// TIA Portal V17 export
// export: Created 2025-03-07T09:23:49.8339125Z, ExportSetting WithDefaults, DisplayName Totally Integrated Automation Portal, DisplayVersion V17 Update 8, DisplayName TIA Portal Openness, DisplayVersion V17 Update 8, DisplayName TIA Portal Version Control Interface, DisplayVersion V17, DisplayName SINAMICS Startdrive Advanced, DisplayVersion V17 SP2, DisplayName SINAMICS Startdrive G110M, G120, G120C, G120D, G120P, G115D, DisplayVersion V17 SP2, DisplayName SINAMICS Startdrive G130, G150, S120, S150, SINAMICS MV, S210, DisplayVersion V17 SP2, DisplayName STEP 7 Professional, DisplayVersion V17 Update 8, DisplayName SINUMERIK ONE STEP 7 Toolbox, DisplayVersion V17 Update 12, DisplayName SINUMERIK 840D sl STEP 7 Toolbox, DisplayVersion V17 Update 12, DisplayName STEP 7 Safety, DisplayVersion V17 Update 6, DisplayName WinCC Advanced, DisplayVersion V17 Update 8
FUNCTION "FC7342_POWDER_TO_MACHINE_INTERLOCK" : Void   // FC7342, LAD
{ S7_Optimized_Access := 'TRUE' }
VERSION : 0.1
// stored: AutoNumber false, IsIECCheckEnabled false, SetENOAutomatically false, UDAEnableTagReadback false
BEGIN

REGION Network 1: LIFE BIT
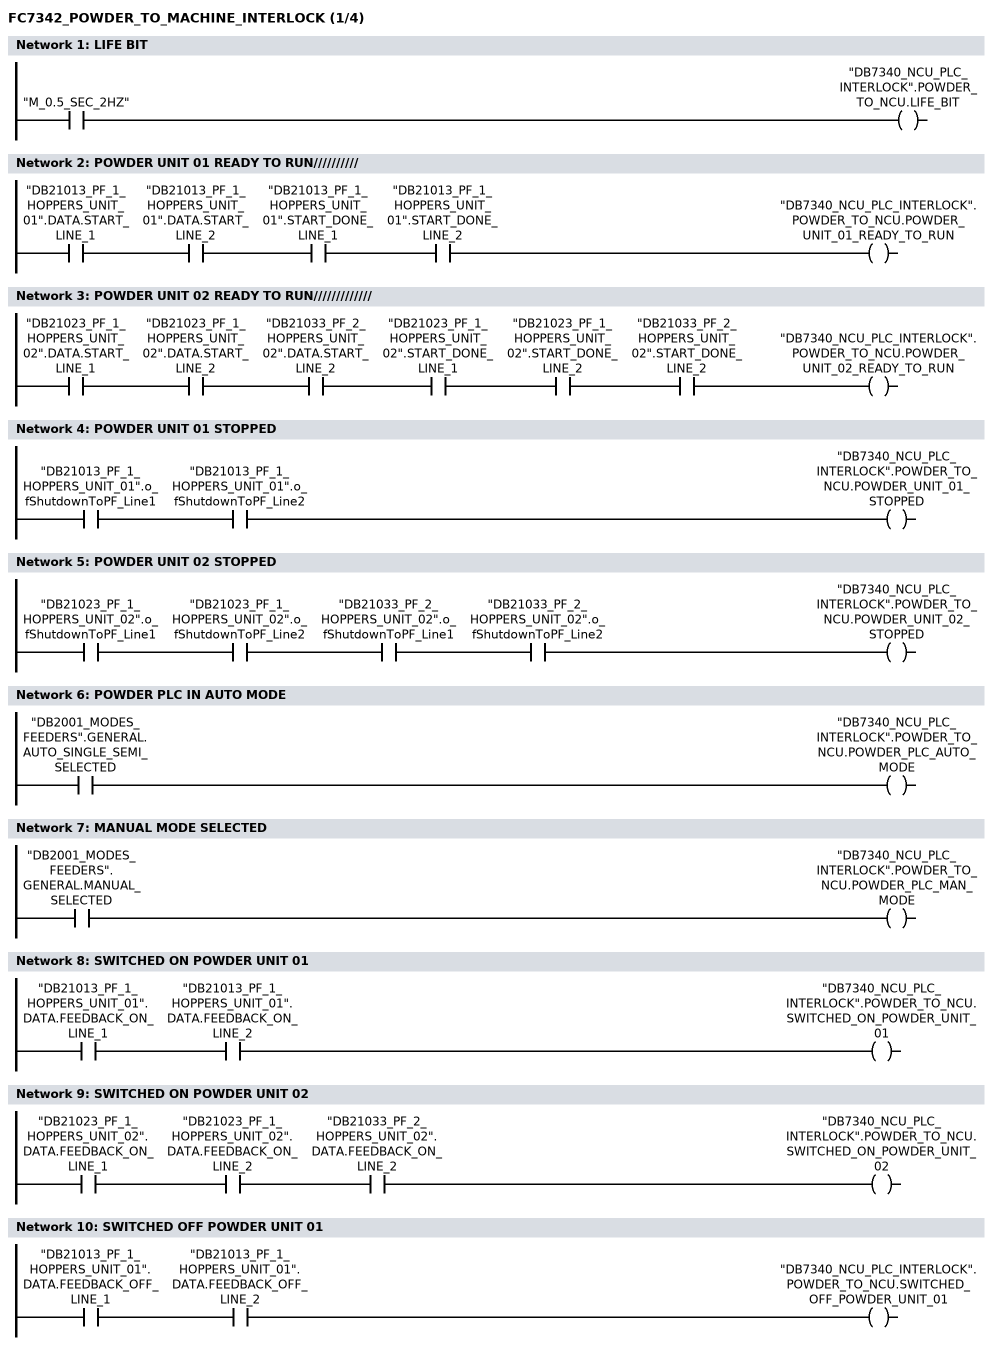
   RUNG wire#powerrail
      Contact( "M_0.5_SEC_2HZ" )
      Coil( "DB7340_NCU_PLC_INTERLOCK".POWDER_TO_NCU.LIFE_BIT )
   END_RUNG
   // the same network as SCL:
   "DB7340_NCU_PLC_INTERLOCK".POWDER_TO_NCU.LIFE_BIT := "M_0.5_SEC_2HZ";
END_REGION

REGION Network 2: POWDER UNIT 01 READY TO RUN//////////
   RUNG wire#powerrail
      Contact( "DB21013_PF_1_HOPPERS_UNIT_01".DATA.START_LINE_1 )
      Contact( "DB21013_PF_1_HOPPERS_UNIT_01".DATA.START_LINE_2 )
      Contact( "DB21013_PF_1_HOPPERS_UNIT_01".START_DONE_LINE_1 )
      Contact( "DB21013_PF_1_HOPPERS_UNIT_01".START_DONE_LINE_2 )
      Coil( "DB7340_NCU_PLC_INTERLOCK".POWDER_TO_NCU.POWDER_UNIT_01_READY_TO_RUN )
   END_RUNG
   // the same network as SCL:
   "DB7340_NCU_PLC_INTERLOCK".POWDER_TO_NCU.POWDER_UNIT_01_READY_TO_RUN := "DB21013_PF_1_HOPPERS_UNIT_01".DATA.START_LINE_1 AND "DB21013_PF_1_HOPPERS_UNIT_01".DATA.START_LINE_2 AND "DB21013_PF_1_HOPPERS_UNIT_01".START_DONE_LINE_1 AND "DB21013_PF_1_HOPPERS_UNIT_01".START_DONE_LINE_2;
END_REGION

REGION Network 3: POWDER UNIT 02 READY TO RUN/////////////
   RUNG wire#powerrail
      Contact( "DB21023_PF_1_HOPPERS_UNIT_02".DATA.START_LINE_1 )
      Contact( "DB21023_PF_1_HOPPERS_UNIT_02".DATA.START_LINE_2 )
      Contact( "DB21033_PF_2_HOPPERS_UNIT_02".DATA.START_LINE_2 )
      Contact( "DB21023_PF_1_HOPPERS_UNIT_02".START_DONE_LINE_1 )
      Contact( "DB21023_PF_1_HOPPERS_UNIT_02".START_DONE_LINE_2 )
      Contact( "DB21033_PF_2_HOPPERS_UNIT_02".START_DONE_LINE_2 )
      Coil( "DB7340_NCU_PLC_INTERLOCK".POWDER_TO_NCU.POWDER_UNIT_02_READY_TO_RUN )
   END_RUNG
   // the same network as SCL:
   "DB7340_NCU_PLC_INTERLOCK".POWDER_TO_NCU.POWDER_UNIT_02_READY_TO_RUN := "DB21023_PF_1_HOPPERS_UNIT_02".DATA.START_LINE_1 AND "DB21023_PF_1_HOPPERS_UNIT_02".DATA.START_LINE_2 AND "DB21033_PF_2_HOPPERS_UNIT_02".DATA.START_LINE_2 AND "DB21023_PF_1_HOPPERS_UNIT_02".START_DONE_LINE_1 AND "DB21023_PF_1_HOPPERS_UNIT_02".START_DONE_LINE_2 AND "DB21033_PF_2_HOPPERS_UNIT_02".START_DONE_LINE_2;
END_REGION

REGION Network 4: POWDER UNIT 01 STOPPED
   RUNG wire#powerrail
      Contact( "DB21013_PF_1_HOPPERS_UNIT_01".o_fShutdownToPF_Line1 )
      Contact( "DB21013_PF_1_HOPPERS_UNIT_01".o_fShutdownToPF_Line2 )
      Coil( "DB7340_NCU_PLC_INTERLOCK".POWDER_TO_NCU.POWDER_UNIT_01_STOPPED )
   END_RUNG
   // the same network as SCL:
   "DB7340_NCU_PLC_INTERLOCK".POWDER_TO_NCU.POWDER_UNIT_01_STOPPED := "DB21013_PF_1_HOPPERS_UNIT_01".o_fShutdownToPF_Line1 AND "DB21013_PF_1_HOPPERS_UNIT_01".o_fShutdownToPF_Line2;
END_REGION

REGION Network 5: POWDER UNIT 02 STOPPED
   RUNG wire#powerrail
      Contact( "DB21023_PF_1_HOPPERS_UNIT_02".o_fShutdownToPF_Line1 )
      Contact( "DB21023_PF_1_HOPPERS_UNIT_02".o_fShutdownToPF_Line2 )
      Contact( "DB21033_PF_2_HOPPERS_UNIT_02".o_fShutdownToPF_Line1 )
      Contact( "DB21033_PF_2_HOPPERS_UNIT_02".o_fShutdownToPF_Line2 )
      Coil( "DB7340_NCU_PLC_INTERLOCK".POWDER_TO_NCU.POWDER_UNIT_02_STOPPED )
   END_RUNG
   // the same network as SCL:
   "DB7340_NCU_PLC_INTERLOCK".POWDER_TO_NCU.POWDER_UNIT_02_STOPPED := "DB21023_PF_1_HOPPERS_UNIT_02".o_fShutdownToPF_Line1 AND "DB21023_PF_1_HOPPERS_UNIT_02".o_fShutdownToPF_Line2 AND "DB21033_PF_2_HOPPERS_UNIT_02".o_fShutdownToPF_Line1 AND "DB21033_PF_2_HOPPERS_UNIT_02".o_fShutdownToPF_Line2;
END_REGION

REGION Network 6: POWDER PLC IN AUTO MODE
   RUNG wire#powerrail
      Contact( "DB2001_MODES_FEEDERS".GENERAL.AUTO_SINGLE_SEMI_SELECTED )
      Coil( "DB7340_NCU_PLC_INTERLOCK".POWDER_TO_NCU.POWDER_PLC_AUTO_MODE )
   END_RUNG
   // the same network as SCL:
   "DB7340_NCU_PLC_INTERLOCK".POWDER_TO_NCU.POWDER_PLC_AUTO_MODE := "DB2001_MODES_FEEDERS".GENERAL.AUTO_SINGLE_SEMI_SELECTED;
END_REGION

REGION Network 7: MANUAL MODE SELECTED
   RUNG wire#powerrail
      Contact( "DB2001_MODES_FEEDERS".GENERAL.MANUAL_SELECTED )
      Coil( "DB7340_NCU_PLC_INTERLOCK".POWDER_TO_NCU.POWDER_PLC_MAN_MODE )
   END_RUNG
   // the same network as SCL:
   "DB7340_NCU_PLC_INTERLOCK".POWDER_TO_NCU.POWDER_PLC_MAN_MODE := "DB2001_MODES_FEEDERS".GENERAL.MANUAL_SELECTED;
END_REGION

REGION Network 8: SWITCHED ON POWDER UNIT 01
   RUNG wire#powerrail
      Contact( "DB21013_PF_1_HOPPERS_UNIT_01".DATA.FEEDBACK_ON_LINE_1 )
      Contact( "DB21013_PF_1_HOPPERS_UNIT_01".DATA.FEEDBACK_ON_LINE_2 )
      Coil( "DB7340_NCU_PLC_INTERLOCK".POWDER_TO_NCU.SWITCHED_ON_POWDER_UNIT_01 )
   END_RUNG
   // the same network as SCL:
   "DB7340_NCU_PLC_INTERLOCK".POWDER_TO_NCU.SWITCHED_ON_POWDER_UNIT_01 := "DB21013_PF_1_HOPPERS_UNIT_01".DATA.FEEDBACK_ON_LINE_1 AND "DB21013_PF_1_HOPPERS_UNIT_01".DATA.FEEDBACK_ON_LINE_2;
END_REGION

REGION Network 9: SWITCHED ON POWDER UNIT 02
   RUNG wire#powerrail
      Contact( "DB21023_PF_1_HOPPERS_UNIT_02".DATA.FEEDBACK_ON_LINE_1 )
      Contact( "DB21023_PF_1_HOPPERS_UNIT_02".DATA.FEEDBACK_ON_LINE_2 )
      Contact( "DB21033_PF_2_HOPPERS_UNIT_02".DATA.FEEDBACK_ON_LINE_2 )
      Coil( "DB7340_NCU_PLC_INTERLOCK".POWDER_TO_NCU.SWITCHED_ON_POWDER_UNIT_02 )
   END_RUNG
   // the same network as SCL:
   "DB7340_NCU_PLC_INTERLOCK".POWDER_TO_NCU.SWITCHED_ON_POWDER_UNIT_02 := "DB21023_PF_1_HOPPERS_UNIT_02".DATA.FEEDBACK_ON_LINE_1 AND "DB21023_PF_1_HOPPERS_UNIT_02".DATA.FEEDBACK_ON_LINE_2 AND "DB21033_PF_2_HOPPERS_UNIT_02".DATA.FEEDBACK_ON_LINE_2;
END_REGION

REGION Network 10: SWITCHED OFF POWDER UNIT 01
   RUNG wire#powerrail
      Contact( "DB21013_PF_1_HOPPERS_UNIT_01".DATA.FEEDBACK_OFF_LINE_1 )
      Contact( "DB21013_PF_1_HOPPERS_UNIT_01".DATA.FEEDBACK_OFF_LINE_2 )
      Coil( "DB7340_NCU_PLC_INTERLOCK".POWDER_TO_NCU.SWITCHED_OFF_POWDER_UNIT_01 )
   END_RUNG
   // the same network as SCL:
   "DB7340_NCU_PLC_INTERLOCK".POWDER_TO_NCU.SWITCHED_OFF_POWDER_UNIT_01 := "DB21013_PF_1_HOPPERS_UNIT_01".DATA.FEEDBACK_OFF_LINE_1 AND "DB21013_PF_1_HOPPERS_UNIT_01".DATA.FEEDBACK_OFF_LINE_2;
END_REGION

REGION Network 11: SWITCHED OFF POWDER UNIT 02
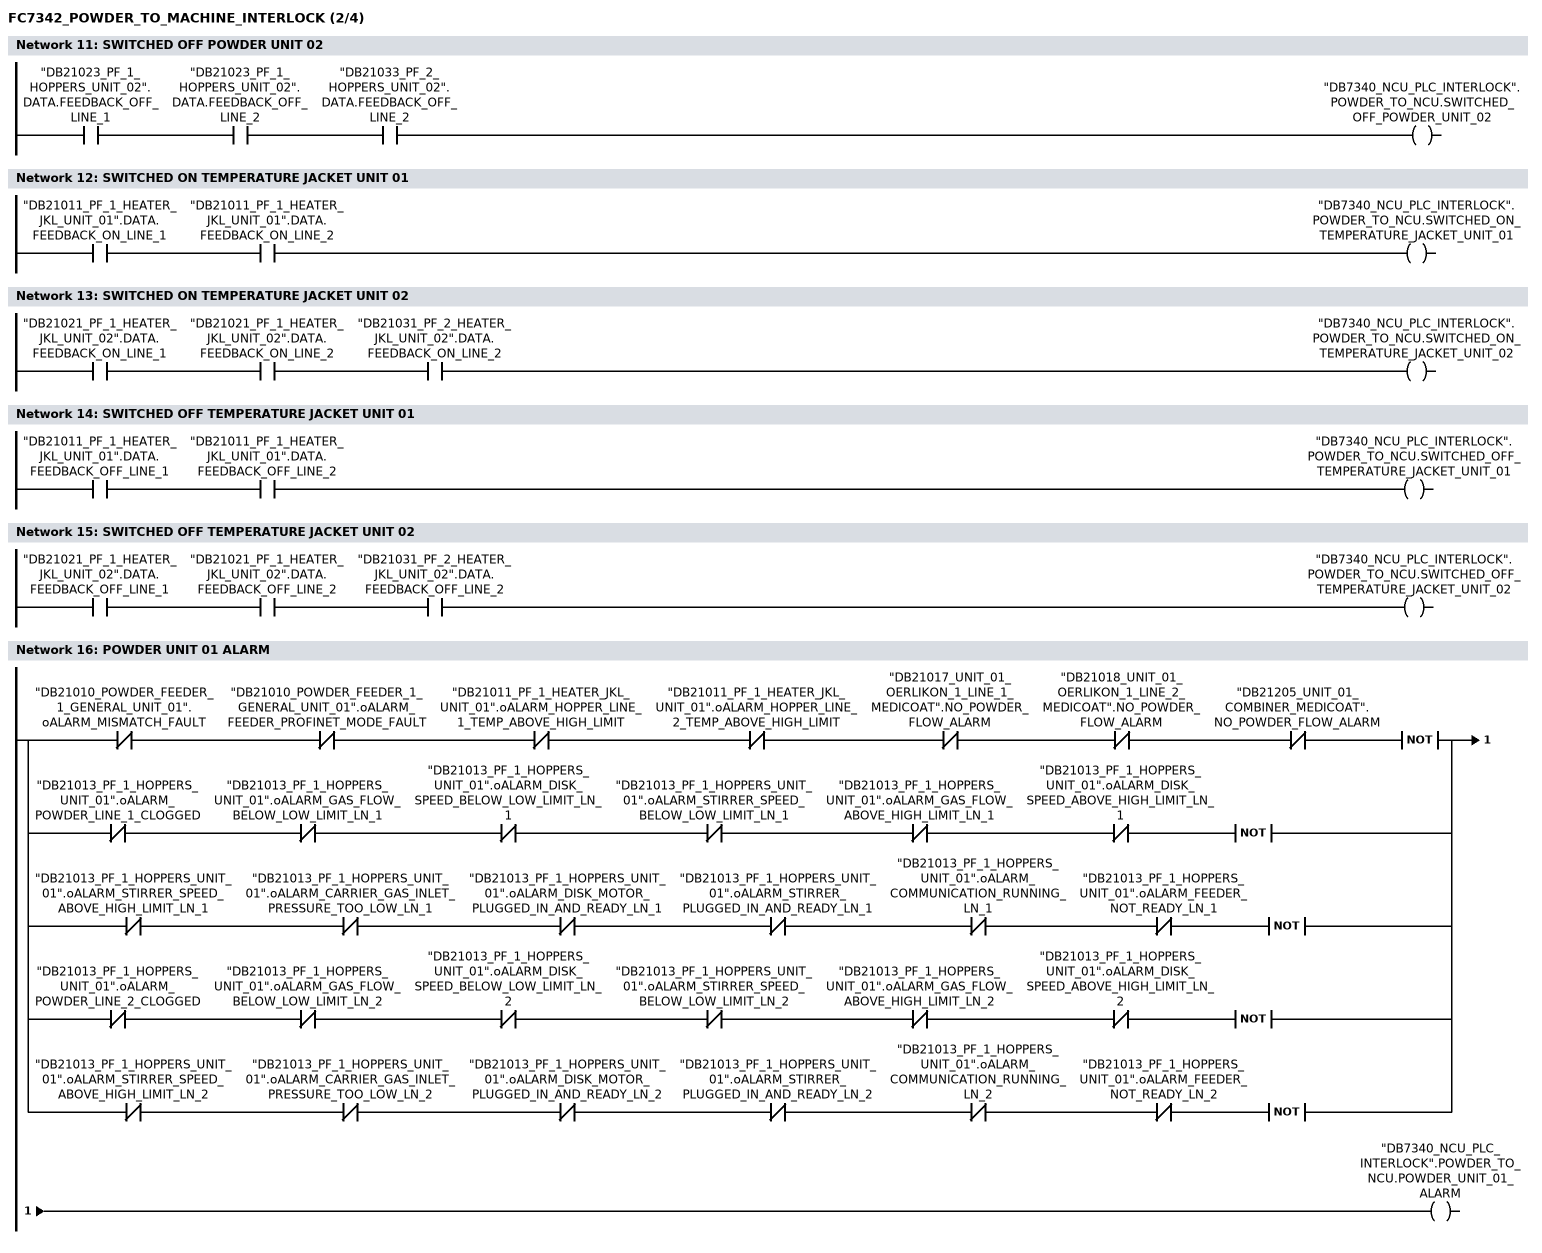
   RUNG wire#powerrail
      Contact( "DB21023_PF_1_HOPPERS_UNIT_02".DATA.FEEDBACK_OFF_LINE_1 )
      Contact( "DB21023_PF_1_HOPPERS_UNIT_02".DATA.FEEDBACK_OFF_LINE_2 )
      Contact( "DB21033_PF_2_HOPPERS_UNIT_02".DATA.FEEDBACK_OFF_LINE_2 )
      Coil( "DB7340_NCU_PLC_INTERLOCK".POWDER_TO_NCU.SWITCHED_OFF_POWDER_UNIT_02 )
   END_RUNG
   // the same network as SCL:
   "DB7340_NCU_PLC_INTERLOCK".POWDER_TO_NCU.SWITCHED_OFF_POWDER_UNIT_02 := "DB21023_PF_1_HOPPERS_UNIT_02".DATA.FEEDBACK_OFF_LINE_1 AND "DB21023_PF_1_HOPPERS_UNIT_02".DATA.FEEDBACK_OFF_LINE_2 AND "DB21033_PF_2_HOPPERS_UNIT_02".DATA.FEEDBACK_OFF_LINE_2;
END_REGION

REGION Network 12: SWITCHED ON TEMPERATURE JACKET UNIT 01
   RUNG wire#powerrail
      Contact( "DB21011_PF_1_HEATER_JKL_UNIT_01".DATA.FEEDBACK_ON_LINE_1 )
      Contact( "DB21011_PF_1_HEATER_JKL_UNIT_01".DATA.FEEDBACK_ON_LINE_2 )
      Coil( "DB7340_NCU_PLC_INTERLOCK".POWDER_TO_NCU.SWITCHED_ON_TEMPERATURE_JACKET_UNIT_01 )
   END_RUNG
   // the same network as SCL:
   "DB7340_NCU_PLC_INTERLOCK".POWDER_TO_NCU.SWITCHED_ON_TEMPERATURE_JACKET_UNIT_01 := "DB21011_PF_1_HEATER_JKL_UNIT_01".DATA.FEEDBACK_ON_LINE_1 AND "DB21011_PF_1_HEATER_JKL_UNIT_01".DATA.FEEDBACK_ON_LINE_2;
END_REGION

REGION Network 13: SWITCHED ON TEMPERATURE JACKET UNIT 02
   RUNG wire#powerrail
      Contact( "DB21021_PF_1_HEATER_JKL_UNIT_02".DATA.FEEDBACK_ON_LINE_1 )
      Contact( "DB21021_PF_1_HEATER_JKL_UNIT_02".DATA.FEEDBACK_ON_LINE_2 )
      Contact( "DB21031_PF_2_HEATER_JKL_UNIT_02".DATA.FEEDBACK_ON_LINE_2 )
      Coil( "DB7340_NCU_PLC_INTERLOCK".POWDER_TO_NCU.SWITCHED_ON_TEMPERATURE_JACKET_UNIT_02 )
   END_RUNG
   // the same network as SCL:
   "DB7340_NCU_PLC_INTERLOCK".POWDER_TO_NCU.SWITCHED_ON_TEMPERATURE_JACKET_UNIT_02 := "DB21021_PF_1_HEATER_JKL_UNIT_02".DATA.FEEDBACK_ON_LINE_1 AND "DB21021_PF_1_HEATER_JKL_UNIT_02".DATA.FEEDBACK_ON_LINE_2 AND "DB21031_PF_2_HEATER_JKL_UNIT_02".DATA.FEEDBACK_ON_LINE_2;
END_REGION

REGION Network 14: SWITCHED OFF TEMPERATURE JACKET UNIT 01
   RUNG wire#powerrail
      Contact( "DB21011_PF_1_HEATER_JKL_UNIT_01".DATA.FEEDBACK_OFF_LINE_1 )
      Contact( "DB21011_PF_1_HEATER_JKL_UNIT_01".DATA.FEEDBACK_OFF_LINE_2 )
      Coil( "DB7340_NCU_PLC_INTERLOCK".POWDER_TO_NCU.SWITCHED_OFF_TEMPERATURE_JACKET_UNIT_01 )
   END_RUNG
   // the same network as SCL:
   "DB7340_NCU_PLC_INTERLOCK".POWDER_TO_NCU.SWITCHED_OFF_TEMPERATURE_JACKET_UNIT_01 := "DB21011_PF_1_HEATER_JKL_UNIT_01".DATA.FEEDBACK_OFF_LINE_1 AND "DB21011_PF_1_HEATER_JKL_UNIT_01".DATA.FEEDBACK_OFF_LINE_2;
END_REGION

REGION Network 15: SWITCHED OFF TEMPERATURE JACKET UNIT 02
   RUNG wire#powerrail
      Contact( "DB21021_PF_1_HEATER_JKL_UNIT_02".DATA.FEEDBACK_OFF_LINE_1 )
      Contact( "DB21021_PF_1_HEATER_JKL_UNIT_02".DATA.FEEDBACK_OFF_LINE_2 )
      Contact( "DB21031_PF_2_HEATER_JKL_UNIT_02".DATA.FEEDBACK_OFF_LINE_2 )
      Coil( "DB7340_NCU_PLC_INTERLOCK".POWDER_TO_NCU.SWITCHED_OFF_TEMPERATURE_JACKET_UNIT_02 )
   END_RUNG
   // the same network as SCL:
   "DB7340_NCU_PLC_INTERLOCK".POWDER_TO_NCU.SWITCHED_OFF_TEMPERATURE_JACKET_UNIT_02 := "DB21021_PF_1_HEATER_JKL_UNIT_02".DATA.FEEDBACK_OFF_LINE_1 AND "DB21021_PF_1_HEATER_JKL_UNIT_02".DATA.FEEDBACK_OFF_LINE_2 AND "DB21031_PF_2_HEATER_JKL_UNIT_02".DATA.FEEDBACK_OFF_LINE_2;
END_REGION

REGION Network 16: POWDER UNIT 01 ALARM
   RUNG wire#powerrail
      I_Contact( "DB21010_POWDER_FEEDER_1_GENERAL_UNIT_01".oALARM_MISMATCH_FAULT )
      I_Contact( "DB21010_POWDER_FEEDER_1_GENERAL_UNIT_01".oALARM_FEEDER_PROFINET_MODE_FAULT )
      I_Contact( "DB21011_PF_1_HEATER_JKL_UNIT_01".oALARM_HOPPER_LINE_1_TEMP_ABOVE_HIGH_LIMIT )
      I_Contact( "DB21011_PF_1_HEATER_JKL_UNIT_01".oALARM_HOPPER_LINE_2_TEMP_ABOVE_HIGH_LIMIT )
      I_Contact( "DB21017_UNIT_01_OERLIKON_1_LINE_1_MEDICOAT".NO_POWDER_FLOW_ALARM )
      I_Contact( "DB21018_UNIT_01_OERLIKON_1_LINE_2_MEDICOAT".NO_POWDER_FLOW_ALARM )
      I_Contact( "DB21205_UNIT_01_COMBINER_MEDICOAT".NO_POWDER_FLOW_ALARM )
      Not()
      wire#w1
      Coil( "DB7340_NCU_PLC_INTERLOCK".POWDER_TO_NCU.POWDER_UNIT_01_ALARM )
   END_RUNG
   RUNG wire#powerrail
      I_Contact( "DB21013_PF_1_HOPPERS_UNIT_01".oALARM_POWDER_LINE_1_CLOGGED )
      I_Contact( "DB21013_PF_1_HOPPERS_UNIT_01".oALARM_GAS_FLOW_BELOW_LOW_LIMIT_LN_1 )
      I_Contact( "DB21013_PF_1_HOPPERS_UNIT_01".oALARM_DISK_SPEED_BELOW_LOW_LIMIT_LN_1 )
      I_Contact( "DB21013_PF_1_HOPPERS_UNIT_01".oALARM_STIRRER_SPEED_BELOW_LOW_LIMIT_LN_1 )
      I_Contact( "DB21013_PF_1_HOPPERS_UNIT_01".oALARM_GAS_FLOW_ABOVE_HIGH_LIMIT_LN_1 )
      I_Contact( "DB21013_PF_1_HOPPERS_UNIT_01".oALARM_DISK_SPEED_ABOVE_HIGH_LIMIT_LN_1 )
      Not()
   END_RUNG wire#w1
   RUNG wire#powerrail
      I_Contact( "DB21013_PF_1_HOPPERS_UNIT_01".oALARM_STIRRER_SPEED_ABOVE_HIGH_LIMIT_LN_1 )
      I_Contact( "DB21013_PF_1_HOPPERS_UNIT_01".oALARM_CARRIER_GAS_INLET_PRESSURE_TOO_LOW_LN_1 )
      I_Contact( "DB21013_PF_1_HOPPERS_UNIT_01".oALARM_DISK_MOTOR_PLUGGED_IN_AND_READY_LN_1 )
      I_Contact( "DB21013_PF_1_HOPPERS_UNIT_01".oALARM_STIRRER_PLUGGED_IN_AND_READY_LN_1 )
      I_Contact( "DB21013_PF_1_HOPPERS_UNIT_01".oALARM_COMMUNICATION_RUNNING_LN_1 )
      I_Contact( "DB21013_PF_1_HOPPERS_UNIT_01".oALARM_FEEDER_NOT_READY_LN_1 )
      Not()
   END_RUNG wire#w1
   RUNG wire#powerrail
      I_Contact( "DB21013_PF_1_HOPPERS_UNIT_01".oALARM_POWDER_LINE_2_CLOGGED )
      I_Contact( "DB21013_PF_1_HOPPERS_UNIT_01".oALARM_GAS_FLOW_BELOW_LOW_LIMIT_LN_2 )
      I_Contact( "DB21013_PF_1_HOPPERS_UNIT_01".oALARM_DISK_SPEED_BELOW_LOW_LIMIT_LN_2 )
      I_Contact( "DB21013_PF_1_HOPPERS_UNIT_01".oALARM_STIRRER_SPEED_BELOW_LOW_LIMIT_LN_2 )
      I_Contact( "DB21013_PF_1_HOPPERS_UNIT_01".oALARM_GAS_FLOW_ABOVE_HIGH_LIMIT_LN_2 )
      I_Contact( "DB21013_PF_1_HOPPERS_UNIT_01".oALARM_DISK_SPEED_ABOVE_HIGH_LIMIT_LN_2 )
      Not()
   END_RUNG wire#w1
   RUNG wire#powerrail
      I_Contact( "DB21013_PF_1_HOPPERS_UNIT_01".oALARM_STIRRER_SPEED_ABOVE_HIGH_LIMIT_LN_2 )
      I_Contact( "DB21013_PF_1_HOPPERS_UNIT_01".oALARM_CARRIER_GAS_INLET_PRESSURE_TOO_LOW_LN_2 )
      I_Contact( "DB21013_PF_1_HOPPERS_UNIT_01".oALARM_DISK_MOTOR_PLUGGED_IN_AND_READY_LN_2 )
      I_Contact( "DB21013_PF_1_HOPPERS_UNIT_01".oALARM_STIRRER_PLUGGED_IN_AND_READY_LN_2 )
      I_Contact( "DB21013_PF_1_HOPPERS_UNIT_01".oALARM_COMMUNICATION_RUNNING_LN_2 )
      I_Contact( "DB21013_PF_1_HOPPERS_UNIT_01".oALARM_FEEDER_NOT_READY_LN_2 )
      Not()
   END_RUNG wire#w1
   // the same network as SCL:
   "DB7340_NCU_PLC_INTERLOCK".POWDER_TO_NCU.POWDER_UNIT_01_ALARM := NOT (NOT "DB21010_POWDER_FEEDER_1_GENERAL_UNIT_01".oALARM_MISMATCH_FAULT AND NOT "DB21010_POWDER_FEEDER_1_GENERAL_UNIT_01".oALARM_FEEDER_PROFINET_MODE_FAULT AND NOT "DB21011_PF_1_HEATER_JKL_UNIT_01".oALARM_HOPPER_LINE_1_TEMP_ABOVE_HIGH_LIMIT AND NOT "DB21011_PF_1_HEATER_JKL_UNIT_01".oALARM_HOPPER_LINE_2_TEMP_ABOVE_HIGH_LIMIT AND NOT "DB21017_UNIT_01_OERLIKON_1_LINE_1_MEDICOAT".NO_POWDER_FLOW_ALARM AND NOT "DB21018_UNIT_01_OERLIKON_1_LINE_2_MEDICOAT".NO_POWDER_FLOW_ALARM AND NOT "DB21205_UNIT_01_COMBINER_MEDICOAT".NO_POWDER_FLOW_ALARM) OR NOT (NOT "DB21013_PF_1_HOPPERS_UNIT_01".oALARM_POWDER_LINE_1_CLOGGED AND NOT "DB21013_PF_1_HOPPERS_UNIT_01".oALARM_GAS_FLOW_BELOW_LOW_LIMIT_LN_1 AND NOT "DB21013_PF_1_HOPPERS_UNIT_01".oALARM_DISK_SPEED_BELOW_LOW_LIMIT_LN_1 AND NOT "DB21013_PF_1_HOPPERS_UNIT_01".oALARM_STIRRER_SPEED_BELOW_LOW_LIMIT_LN_1 AND NOT "DB21013_PF_1_HOPPERS_UNIT_01".oALARM_GAS_FLOW_ABOVE_HIGH_LIMIT_LN_1 AND NOT "DB21013_PF_1_HOPPERS_UNIT_01".oALARM_DISK_SPEED_ABOVE_HIGH_LIMIT_LN_1) OR NOT (NOT "DB21013_PF_1_HOPPERS_UNIT_01".oALARM_STIRRER_SPEED_ABOVE_HIGH_LIMIT_LN_1 AND NOT "DB21013_PF_1_HOPPERS_UNIT_01".oALARM_CARRIER_GAS_INLET_PRESSURE_TOO_LOW_LN_1 AND NOT "DB21013_PF_1_HOPPERS_UNIT_01".oALARM_DISK_MOTOR_PLUGGED_IN_AND_READY_LN_1 AND NOT "DB21013_PF_1_HOPPERS_UNIT_01".oALARM_STIRRER_PLUGGED_IN_AND_READY_LN_1 AND NOT "DB21013_PF_1_HOPPERS_UNIT_01".oALARM_COMMUNICATION_RUNNING_LN_1 AND NOT "DB21013_PF_1_HOPPERS_UNIT_01".oALARM_FEEDER_NOT_READY_LN_1) OR NOT (NOT "DB21013_PF_1_HOPPERS_UNIT_01".oALARM_POWDER_LINE_2_CLOGGED AND NOT "DB21013_PF_1_HOPPERS_UNIT_01".oALARM_GAS_FLOW_BELOW_LOW_LIMIT_LN_2 AND NOT "DB21013_PF_1_HOPPERS_UNIT_01".oALARM_DISK_SPEED_BELOW_LOW_LIMIT_LN_2 AND NOT "DB21013_PF_1_HOPPERS_UNIT_01".oALARM_STIRRER_SPEED_BELOW_LOW_LIMIT_LN_2 AND NOT "DB21013_PF_1_HOPPERS_UNIT_01".oALARM_GAS_FLOW_ABOVE_HIGH_LIMIT_LN_2 AND NOT "DB21013_PF_1_HOPPERS_UNIT_01".oALARM_DISK_SPEED_ABOVE_HIGH_LIMIT_LN_2) OR NOT (NOT "DB21013_PF_1_HOPPERS_UNIT_01".oALARM_STIRRER_SPEED_ABOVE_HIGH_LIMIT_LN_2 AND NOT "DB21013_PF_1_HOPPERS_UNIT_01".oALARM_CARRIER_GAS_INLET_PRESSURE_TOO_LOW_LN_2 AND NOT "DB21013_PF_1_HOPPERS_UNIT_01".oALARM_DISK_MOTOR_PLUGGED_IN_AND_READY_LN_2 AND NOT "DB21013_PF_1_HOPPERS_UNIT_01".oALARM_STIRRER_PLUGGED_IN_AND_READY_LN_2 AND NOT "DB21013_PF_1_HOPPERS_UNIT_01".oALARM_COMMUNICATION_RUNNING_LN_2 AND NOT "DB21013_PF_1_HOPPERS_UNIT_01".oALARM_FEEDER_NOT_READY_LN_2);
END_REGION

REGION Network 17: POWDER UNIT 02 ALARM
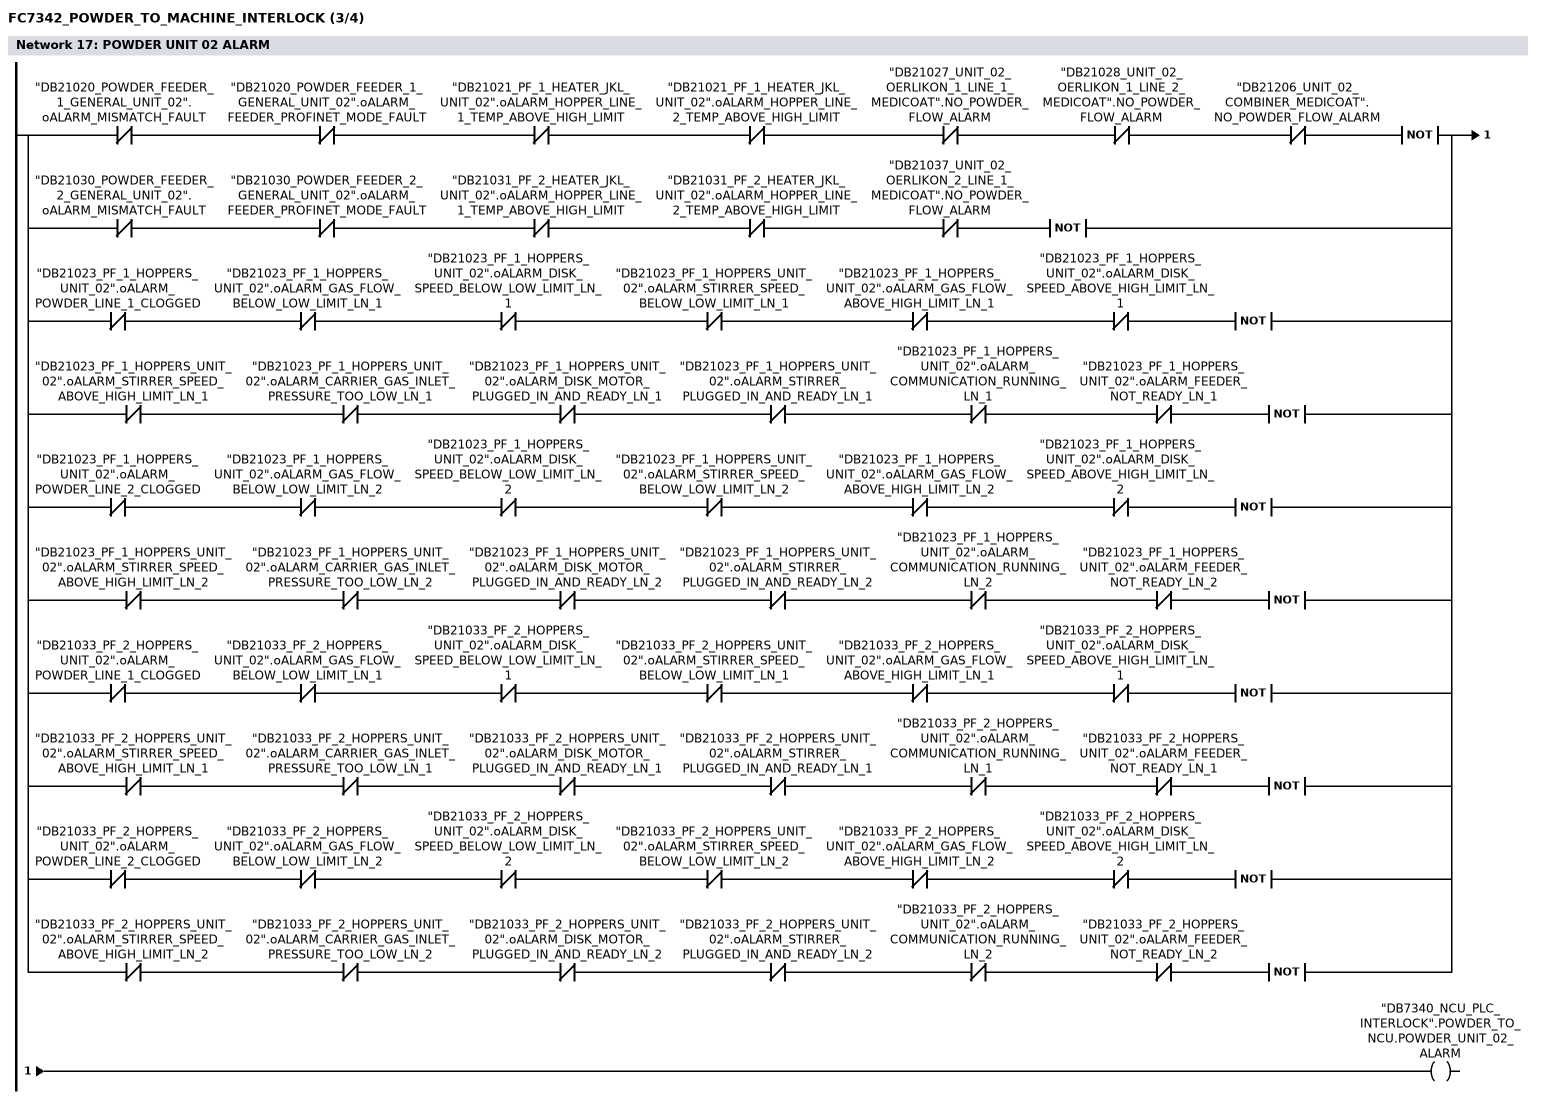
   RUNG wire#powerrail
      I_Contact( "DB21020_POWDER_FEEDER_1_GENERAL_UNIT_02".oALARM_MISMATCH_FAULT )
      I_Contact( "DB21020_POWDER_FEEDER_1_GENERAL_UNIT_02".oALARM_FEEDER_PROFINET_MODE_FAULT )
      I_Contact( "DB21021_PF_1_HEATER_JKL_UNIT_02".oALARM_HOPPER_LINE_1_TEMP_ABOVE_HIGH_LIMIT )
      I_Contact( "DB21021_PF_1_HEATER_JKL_UNIT_02".oALARM_HOPPER_LINE_2_TEMP_ABOVE_HIGH_LIMIT )
      I_Contact( "DB21027_UNIT_02_OERLIKON_1_LINE_1_MEDICOAT".NO_POWDER_FLOW_ALARM )
      I_Contact( "DB21028_UNIT_02_OERLIKON_1_LINE_2_MEDICOAT".NO_POWDER_FLOW_ALARM )
      I_Contact( "DB21206_UNIT_02_COMBINER_MEDICOAT".NO_POWDER_FLOW_ALARM )
      Not()
      wire#w1
      Coil( "DB7340_NCU_PLC_INTERLOCK".POWDER_TO_NCU.POWDER_UNIT_02_ALARM )
   END_RUNG
   RUNG wire#powerrail
      I_Contact( "DB21030_POWDER_FEEDER_2_GENERAL_UNIT_02".oALARM_MISMATCH_FAULT )
      I_Contact( "DB21030_POWDER_FEEDER_2_GENERAL_UNIT_02".oALARM_FEEDER_PROFINET_MODE_FAULT )
      I_Contact( "DB21031_PF_2_HEATER_JKL_UNIT_02".oALARM_HOPPER_LINE_1_TEMP_ABOVE_HIGH_LIMIT )
      I_Contact( "DB21031_PF_2_HEATER_JKL_UNIT_02".oALARM_HOPPER_LINE_2_TEMP_ABOVE_HIGH_LIMIT )
      I_Contact( "DB21037_UNIT_02_OERLIKON_2_LINE_1_MEDICOAT".NO_POWDER_FLOW_ALARM )
      Not()
   END_RUNG wire#w1
   RUNG wire#powerrail
      I_Contact( "DB21023_PF_1_HOPPERS_UNIT_02".oALARM_POWDER_LINE_1_CLOGGED )
      I_Contact( "DB21023_PF_1_HOPPERS_UNIT_02".oALARM_GAS_FLOW_BELOW_LOW_LIMIT_LN_1 )
      I_Contact( "DB21023_PF_1_HOPPERS_UNIT_02".oALARM_DISK_SPEED_BELOW_LOW_LIMIT_LN_1 )
      I_Contact( "DB21023_PF_1_HOPPERS_UNIT_02".oALARM_STIRRER_SPEED_BELOW_LOW_LIMIT_LN_1 )
      I_Contact( "DB21023_PF_1_HOPPERS_UNIT_02".oALARM_GAS_FLOW_ABOVE_HIGH_LIMIT_LN_1 )
      I_Contact( "DB21023_PF_1_HOPPERS_UNIT_02".oALARM_DISK_SPEED_ABOVE_HIGH_LIMIT_LN_1 )
      Not()
   END_RUNG wire#w1
   RUNG wire#powerrail
      I_Contact( "DB21023_PF_1_HOPPERS_UNIT_02".oALARM_STIRRER_SPEED_ABOVE_HIGH_LIMIT_LN_1 )
      I_Contact( "DB21023_PF_1_HOPPERS_UNIT_02".oALARM_CARRIER_GAS_INLET_PRESSURE_TOO_LOW_LN_1 )
      I_Contact( "DB21023_PF_1_HOPPERS_UNIT_02".oALARM_DISK_MOTOR_PLUGGED_IN_AND_READY_LN_1 )
      I_Contact( "DB21023_PF_1_HOPPERS_UNIT_02".oALARM_STIRRER_PLUGGED_IN_AND_READY_LN_1 )
      I_Contact( "DB21023_PF_1_HOPPERS_UNIT_02".oALARM_COMMUNICATION_RUNNING_LN_1 )
      I_Contact( "DB21023_PF_1_HOPPERS_UNIT_02".oALARM_FEEDER_NOT_READY_LN_1 )
      Not()
   END_RUNG wire#w1
   RUNG wire#powerrail
      I_Contact( "DB21023_PF_1_HOPPERS_UNIT_02".oALARM_POWDER_LINE_2_CLOGGED )
      I_Contact( "DB21023_PF_1_HOPPERS_UNIT_02".oALARM_GAS_FLOW_BELOW_LOW_LIMIT_LN_2 )
      I_Contact( "DB21023_PF_1_HOPPERS_UNIT_02".oALARM_DISK_SPEED_BELOW_LOW_LIMIT_LN_2 )
      I_Contact( "DB21023_PF_1_HOPPERS_UNIT_02".oALARM_STIRRER_SPEED_BELOW_LOW_LIMIT_LN_2 )
      I_Contact( "DB21023_PF_1_HOPPERS_UNIT_02".oALARM_GAS_FLOW_ABOVE_HIGH_LIMIT_LN_2 )
      I_Contact( "DB21023_PF_1_HOPPERS_UNIT_02".oALARM_DISK_SPEED_ABOVE_HIGH_LIMIT_LN_2 )
      Not()
   END_RUNG wire#w1
   RUNG wire#powerrail
      I_Contact( "DB21023_PF_1_HOPPERS_UNIT_02".oALARM_STIRRER_SPEED_ABOVE_HIGH_LIMIT_LN_2 )
      I_Contact( "DB21023_PF_1_HOPPERS_UNIT_02".oALARM_CARRIER_GAS_INLET_PRESSURE_TOO_LOW_LN_2 )
      I_Contact( "DB21023_PF_1_HOPPERS_UNIT_02".oALARM_DISK_MOTOR_PLUGGED_IN_AND_READY_LN_2 )
      I_Contact( "DB21023_PF_1_HOPPERS_UNIT_02".oALARM_STIRRER_PLUGGED_IN_AND_READY_LN_2 )
      I_Contact( "DB21023_PF_1_HOPPERS_UNIT_02".oALARM_COMMUNICATION_RUNNING_LN_2 )
      I_Contact( "DB21023_PF_1_HOPPERS_UNIT_02".oALARM_FEEDER_NOT_READY_LN_2 )
      Not()
   END_RUNG wire#w1
   RUNG wire#powerrail
      I_Contact( "DB21033_PF_2_HOPPERS_UNIT_02".oALARM_POWDER_LINE_1_CLOGGED )
      I_Contact( "DB21033_PF_2_HOPPERS_UNIT_02".oALARM_GAS_FLOW_BELOW_LOW_LIMIT_LN_1 )
      I_Contact( "DB21033_PF_2_HOPPERS_UNIT_02".oALARM_DISK_SPEED_BELOW_LOW_LIMIT_LN_1 )
      I_Contact( "DB21033_PF_2_HOPPERS_UNIT_02".oALARM_STIRRER_SPEED_BELOW_LOW_LIMIT_LN_1 )
      I_Contact( "DB21033_PF_2_HOPPERS_UNIT_02".oALARM_GAS_FLOW_ABOVE_HIGH_LIMIT_LN_1 )
      I_Contact( "DB21033_PF_2_HOPPERS_UNIT_02".oALARM_DISK_SPEED_ABOVE_HIGH_LIMIT_LN_1 )
      Not()
   END_RUNG wire#w1
   RUNG wire#powerrail
      I_Contact( "DB21033_PF_2_HOPPERS_UNIT_02".oALARM_STIRRER_SPEED_ABOVE_HIGH_LIMIT_LN_1 )
      I_Contact( "DB21033_PF_2_HOPPERS_UNIT_02".oALARM_CARRIER_GAS_INLET_PRESSURE_TOO_LOW_LN_1 )
      I_Contact( "DB21033_PF_2_HOPPERS_UNIT_02".oALARM_DISK_MOTOR_PLUGGED_IN_AND_READY_LN_1 )
      I_Contact( "DB21033_PF_2_HOPPERS_UNIT_02".oALARM_STIRRER_PLUGGED_IN_AND_READY_LN_1 )
      I_Contact( "DB21033_PF_2_HOPPERS_UNIT_02".oALARM_COMMUNICATION_RUNNING_LN_1 )
      I_Contact( "DB21033_PF_2_HOPPERS_UNIT_02".oALARM_FEEDER_NOT_READY_LN_1 )
      Not()
   END_RUNG wire#w1
   RUNG wire#powerrail
      I_Contact( "DB21033_PF_2_HOPPERS_UNIT_02".oALARM_POWDER_LINE_2_CLOGGED )
      I_Contact( "DB21033_PF_2_HOPPERS_UNIT_02".oALARM_GAS_FLOW_BELOW_LOW_LIMIT_LN_2 )
      I_Contact( "DB21033_PF_2_HOPPERS_UNIT_02".oALARM_DISK_SPEED_BELOW_LOW_LIMIT_LN_2 )
      I_Contact( "DB21033_PF_2_HOPPERS_UNIT_02".oALARM_STIRRER_SPEED_BELOW_LOW_LIMIT_LN_2 )
      I_Contact( "DB21033_PF_2_HOPPERS_UNIT_02".oALARM_GAS_FLOW_ABOVE_HIGH_LIMIT_LN_2 )
      I_Contact( "DB21033_PF_2_HOPPERS_UNIT_02".oALARM_DISK_SPEED_ABOVE_HIGH_LIMIT_LN_2 )
      Not()
   END_RUNG wire#w1
   RUNG wire#powerrail
      I_Contact( "DB21033_PF_2_HOPPERS_UNIT_02".oALARM_STIRRER_SPEED_ABOVE_HIGH_LIMIT_LN_2 )
      I_Contact( "DB21033_PF_2_HOPPERS_UNIT_02".oALARM_CARRIER_GAS_INLET_PRESSURE_TOO_LOW_LN_2 )
      I_Contact( "DB21033_PF_2_HOPPERS_UNIT_02".oALARM_DISK_MOTOR_PLUGGED_IN_AND_READY_LN_2 )
      I_Contact( "DB21033_PF_2_HOPPERS_UNIT_02".oALARM_STIRRER_PLUGGED_IN_AND_READY_LN_2 )
      I_Contact( "DB21033_PF_2_HOPPERS_UNIT_02".oALARM_COMMUNICATION_RUNNING_LN_2 )
      I_Contact( "DB21033_PF_2_HOPPERS_UNIT_02".oALARM_FEEDER_NOT_READY_LN_2 )
      Not()
   END_RUNG wire#w1
   // the same network as SCL:
   "DB7340_NCU_PLC_INTERLOCK".POWDER_TO_NCU.POWDER_UNIT_02_ALARM := NOT (NOT "DB21020_POWDER_FEEDER_1_GENERAL_UNIT_02".oALARM_MISMATCH_FAULT AND NOT "DB21020_POWDER_FEEDER_1_GENERAL_UNIT_02".oALARM_FEEDER_PROFINET_MODE_FAULT AND NOT "DB21021_PF_1_HEATER_JKL_UNIT_02".oALARM_HOPPER_LINE_1_TEMP_ABOVE_HIGH_LIMIT AND NOT "DB21021_PF_1_HEATER_JKL_UNIT_02".oALARM_HOPPER_LINE_2_TEMP_ABOVE_HIGH_LIMIT AND NOT "DB21027_UNIT_02_OERLIKON_1_LINE_1_MEDICOAT".NO_POWDER_FLOW_ALARM AND NOT "DB21028_UNIT_02_OERLIKON_1_LINE_2_MEDICOAT".NO_POWDER_FLOW_ALARM AND NOT "DB21206_UNIT_02_COMBINER_MEDICOAT".NO_POWDER_FLOW_ALARM) OR NOT (NOT "DB21030_POWDER_FEEDER_2_GENERAL_UNIT_02".oALARM_MISMATCH_FAULT AND NOT "DB21030_POWDER_FEEDER_2_GENERAL_UNIT_02".oALARM_FEEDER_PROFINET_MODE_FAULT AND NOT "DB21031_PF_2_HEATER_JKL_UNIT_02".oALARM_HOPPER_LINE_1_TEMP_ABOVE_HIGH_LIMIT AND NOT "DB21031_PF_2_HEATER_JKL_UNIT_02".oALARM_HOPPER_LINE_2_TEMP_ABOVE_HIGH_LIMIT AND NOT "DB21037_UNIT_02_OERLIKON_2_LINE_1_MEDICOAT".NO_POWDER_FLOW_ALARM) OR NOT (NOT "DB21023_PF_1_HOPPERS_UNIT_02".oALARM_POWDER_LINE_1_CLOGGED AND NOT "DB21023_PF_1_HOPPERS_UNIT_02".oALARM_GAS_FLOW_BELOW_LOW_LIMIT_LN_1 AND NOT "DB21023_PF_1_HOPPERS_UNIT_02".oALARM_DISK_SPEED_BELOW_LOW_LIMIT_LN_1 AND NOT "DB21023_PF_1_HOPPERS_UNIT_02".oALARM_STIRRER_SPEED_BELOW_LOW_LIMIT_LN_1 AND NOT "DB21023_PF_1_HOPPERS_UNIT_02".oALARM_GAS_FLOW_ABOVE_HIGH_LIMIT_LN_1 AND NOT "DB21023_PF_1_HOPPERS_UNIT_02".oALARM_DISK_SPEED_ABOVE_HIGH_LIMIT_LN_1) OR NOT (NOT "DB21023_PF_1_HOPPERS_UNIT_02".oALARM_STIRRER_SPEED_ABOVE_HIGH_LIMIT_LN_1 AND NOT "DB21023_PF_1_HOPPERS_UNIT_02".oALARM_CARRIER_GAS_INLET_PRESSURE_TOO_LOW_LN_1 AND NOT "DB21023_PF_1_HOPPERS_UNIT_02".oALARM_DISK_MOTOR_PLUGGED_IN_AND_READY_LN_1 AND NOT "DB21023_PF_1_HOPPERS_UNIT_02".oALARM_STIRRER_PLUGGED_IN_AND_READY_LN_1 AND NOT "DB21023_PF_1_HOPPERS_UNIT_02".oALARM_COMMUNICATION_RUNNING_LN_1 AND NOT "DB21023_PF_1_HOPPERS_UNIT_02".oALARM_FEEDER_NOT_READY_LN_1) OR NOT (NOT "DB21023_PF_1_HOPPERS_UNIT_02".oALARM_POWDER_LINE_2_CLOGGED AND NOT "DB21023_PF_1_HOPPERS_UNIT_02".oALARM_GAS_FLOW_BELOW_LOW_LIMIT_LN_2 AND NOT "DB21023_PF_1_HOPPERS_UNIT_02".oALARM_DISK_SPEED_BELOW_LOW_LIMIT_LN_2 AND NOT "DB21023_PF_1_HOPPERS_UNIT_02".oALARM_STIRRER_SPEED_BELOW_LOW_LIMIT_LN_2 AND NOT "DB21023_PF_1_HOPPERS_UNIT_02".oALARM_GAS_FLOW_ABOVE_HIGH_LIMIT_LN_2 AND NOT "DB21023_PF_1_HOPPERS_UNIT_02".oALARM_DISK_SPEED_ABOVE_HIGH_LIMIT_LN_2) OR NOT (NOT "DB21023_PF_1_HOPPERS_UNIT_02".oALARM_STIRRER_SPEED_ABOVE_HIGH_LIMIT_LN_2 AND NOT "DB21023_PF_1_HOPPERS_UNIT_02".oALARM_CARRIER_GAS_INLET_PRESSURE_TOO_LOW_LN_2 AND NOT "DB21023_PF_1_HOPPERS_UNIT_02".oALARM_DISK_MOTOR_PLUGGED_IN_AND_READY_LN_2 AND NOT "DB21023_PF_1_HOPPERS_UNIT_02".oALARM_STIRRER_PLUGGED_IN_AND_READY_LN_2 AND NOT "DB21023_PF_1_HOPPERS_UNIT_02".oALARM_COMMUNICATION_RUNNING_LN_2 AND NOT "DB21023_PF_1_HOPPERS_UNIT_02".oALARM_FEEDER_NOT_READY_LN_2) OR NOT (NOT "DB21033_PF_2_HOPPERS_UNIT_02".oALARM_POWDER_LINE_1_CLOGGED AND NOT "DB21033_PF_2_HOPPERS_UNIT_02".oALARM_GAS_FLOW_BELOW_LOW_LIMIT_LN_1 AND NOT "DB21033_PF_2_HOPPERS_UNIT_02".oALARM_DISK_SPEED_BELOW_LOW_LIMIT_LN_1 AND NOT "DB21033_PF_2_HOPPERS_UNIT_02".oALARM_STIRRER_SPEED_BELOW_LOW_LIMIT_LN_1 AND NOT "DB21033_PF_2_HOPPERS_UNIT_02".oALARM_GAS_FLOW_ABOVE_HIGH_LIMIT_LN_1 AND NOT "DB21033_PF_2_HOPPERS_UNIT_02".oALARM_DISK_SPEED_ABOVE_HIGH_LIMIT_LN_1) OR NOT (NOT "DB21033_PF_2_HOPPERS_UNIT_02".oALARM_STIRRER_SPEED_ABOVE_HIGH_LIMIT_LN_1 AND NOT "DB21033_PF_2_HOPPERS_UNIT_02".oALARM_CARRIER_GAS_INLET_PRESSURE_TOO_LOW_LN_1 AND NOT "DB21033_PF_2_HOPPERS_UNIT_02".oALARM_DISK_MOTOR_PLUGGED_IN_AND_READY_LN_1 AND NOT "DB21033_PF_2_HOPPERS_UNIT_02".oALARM_STIRRER_PLUGGED_IN_AND_READY_LN_1 AND NOT "DB21033_PF_2_HOPPERS_UNIT_02".oALARM_COMMUNICATION_RUNNING_LN_1 AND NOT "DB21033_PF_2_HOPPERS_UNIT_02".oALARM_FEEDER_NOT_READY_LN_1) OR NOT (NOT "DB21033_PF_2_HOPPERS_UNIT_02".oALARM_POWDER_LINE_2_CLOGGED AND NOT "DB21033_PF_2_HOPPERS_UNIT_02".oALARM_GAS_FLOW_BELOW_LOW_LIMIT_LN_2 AND NOT "DB21033_PF_2_HOPPERS_UNIT_02".oALARM_DISK_SPEED_BELOW_LOW_LIMIT_LN_2 AND NOT "DB21033_PF_2_HOPPERS_UNIT_02".oALARM_STIRRER_SPEED_BELOW_LOW_LIMIT_LN_2 AND NOT "DB21033_PF_2_HOPPERS_UNIT_02".oALARM_GAS_FLOW_ABOVE_HIGH_LIMIT_LN_2 AND NOT "DB21033_PF_2_HOPPERS_UNIT_02".oALARM_DISK_SPEED_ABOVE_HIGH_LIMIT_LN_2) OR NOT (NOT "DB21033_PF_2_HOPPERS_UNIT_02".oALARM_STIRRER_SPEED_ABOVE_HIGH_LIMIT_LN_2 AND NOT "DB21033_PF_2_HOPPERS_UNIT_02".oALARM_CARRIER_GAS_INLET_PRESSURE_TOO_LOW_LN_2 AND NOT "DB21033_PF_2_HOPPERS_UNIT_02".oALARM_DISK_MOTOR_PLUGGED_IN_AND_READY_LN_2 AND NOT "DB21033_PF_2_HOPPERS_UNIT_02".oALARM_STIRRER_PLUGGED_IN_AND_READY_LN_2 AND NOT "DB21033_PF_2_HOPPERS_UNIT_02".oALARM_COMMUNICATION_RUNNING_LN_2 AND NOT "DB21033_PF_2_HOPPERS_UNIT_02".oALARM_FEEDER_NOT_READY_LN_2);
END_REGION

REGION Network 18: UNIT 01 POWDER FEEDER 1 ACTUAL VALUES
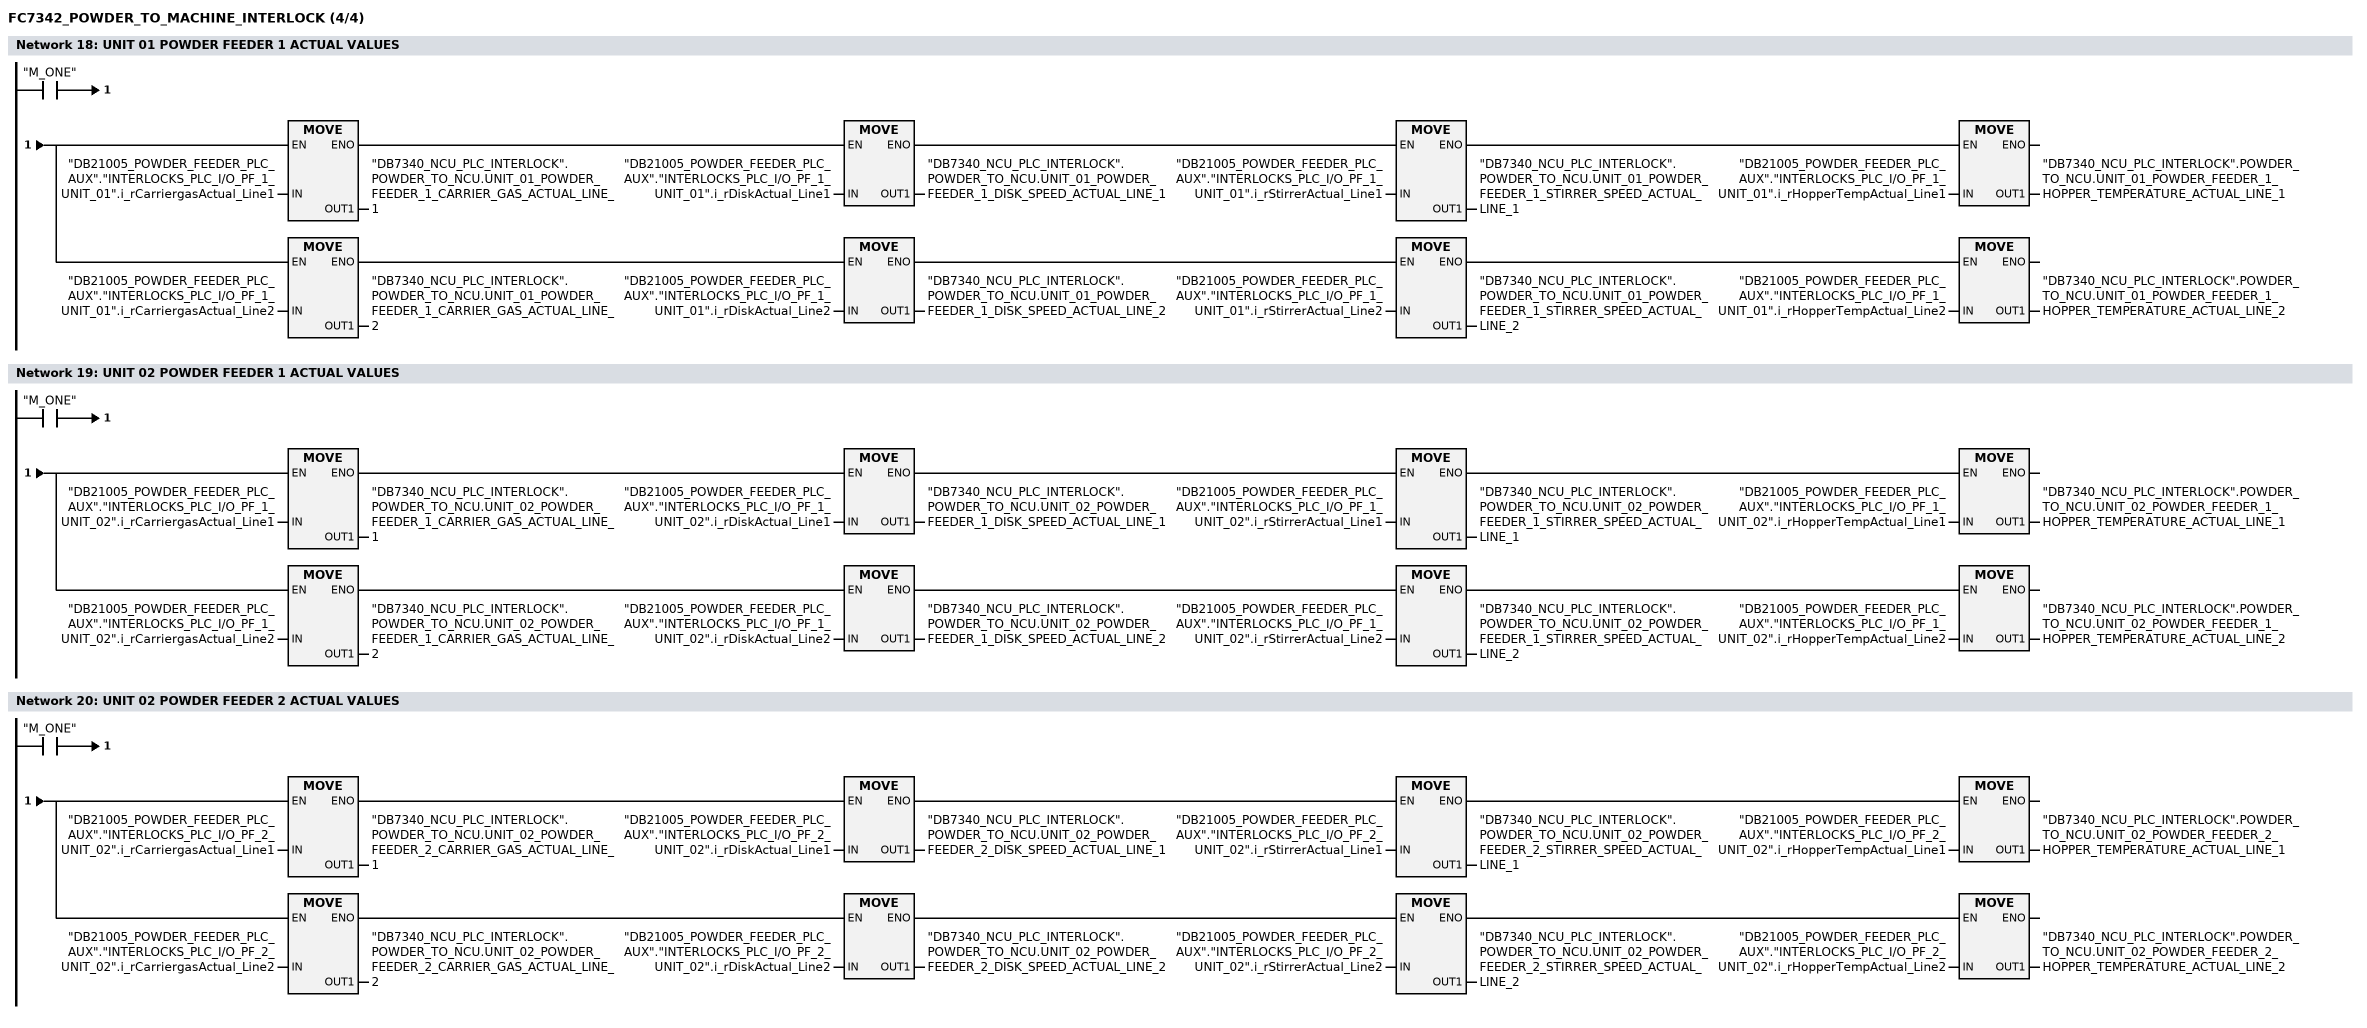
   RUNG wire#powerrail
      Contact( "M_ONE" )
      wire#w1
      Move(in := "DB21005_POWDER_FEEDER_PLC_AUX"."INTERLOCKS_PLC_I/O_PF_1_UNIT_01".i_rCarriergasActual_Line1, out1 => "DB7340_NCU_PLC_INTERLOCK".POWDER_TO_NCU.UNIT_01_POWDER_FEEDER_1_CARRIER_GAS_ACTUAL_LINE_1)
      Move(in := "DB21005_POWDER_FEEDER_PLC_AUX"."INTERLOCKS_PLC_I/O_PF_1_UNIT_01".i_rDiskActual_Line1, out1 => "DB7340_NCU_PLC_INTERLOCK".POWDER_TO_NCU.UNIT_01_POWDER_FEEDER_1_DISK_SPEED_ACTUAL_LINE_1)
      Move(in := "DB21005_POWDER_FEEDER_PLC_AUX"."INTERLOCKS_PLC_I/O_PF_1_UNIT_01".i_rStirrerActual_Line1, out1 => "DB7340_NCU_PLC_INTERLOCK".POWDER_TO_NCU.UNIT_01_POWDER_FEEDER_1_STIRRER_SPEED_ACTUAL_LINE_1)
      Move(in := "DB21005_POWDER_FEEDER_PLC_AUX"."INTERLOCKS_PLC_I/O_PF_1_UNIT_01".i_rHopperTempActual_Line1, out1 => "DB7340_NCU_PLC_INTERLOCK".POWDER_TO_NCU.UNIT_01_POWDER_FEEDER_1_HOPPER_TEMPERATURE_ACTUAL_LINE_1)
   END_RUNG
   RUNG wire#w1
      Move(in := "DB21005_POWDER_FEEDER_PLC_AUX"."INTERLOCKS_PLC_I/O_PF_1_UNIT_01".i_rCarriergasActual_Line2, out1 => "DB7340_NCU_PLC_INTERLOCK".POWDER_TO_NCU.UNIT_01_POWDER_FEEDER_1_CARRIER_GAS_ACTUAL_LINE_2)
      Move(in := "DB21005_POWDER_FEEDER_PLC_AUX"."INTERLOCKS_PLC_I/O_PF_1_UNIT_01".i_rDiskActual_Line2, out1 => "DB7340_NCU_PLC_INTERLOCK".POWDER_TO_NCU.UNIT_01_POWDER_FEEDER_1_DISK_SPEED_ACTUAL_LINE_2)
      Move(in := "DB21005_POWDER_FEEDER_PLC_AUX"."INTERLOCKS_PLC_I/O_PF_1_UNIT_01".i_rStirrerActual_Line2, out1 => "DB7340_NCU_PLC_INTERLOCK".POWDER_TO_NCU.UNIT_01_POWDER_FEEDER_1_STIRRER_SPEED_ACTUAL_LINE_2)
      Move(in := "DB21005_POWDER_FEEDER_PLC_AUX"."INTERLOCKS_PLC_I/O_PF_1_UNIT_01".i_rHopperTempActual_Line2, out1 => "DB7340_NCU_PLC_INTERLOCK".POWDER_TO_NCU.UNIT_01_POWDER_FEEDER_1_HOPPER_TEMPERATURE_ACTUAL_LINE_2)
   END_RUNG
   // the same network as SCL:
   IF "M_ONE" THEN
       "DB7340_NCU_PLC_INTERLOCK".POWDER_TO_NCU.UNIT_01_POWDER_FEEDER_1_CARRIER_GAS_ACTUAL_LINE_1 := "DB21005_POWDER_FEEDER_PLC_AUX"."INTERLOCKS_PLC_I/O_PF_1_UNIT_01".i_rCarriergasActual_Line1;
       "DB7340_NCU_PLC_INTERLOCK".POWDER_TO_NCU.UNIT_01_POWDER_FEEDER_1_DISK_SPEED_ACTUAL_LINE_1 := "DB21005_POWDER_FEEDER_PLC_AUX"."INTERLOCKS_PLC_I/O_PF_1_UNIT_01".i_rDiskActual_Line1;
       "DB7340_NCU_PLC_INTERLOCK".POWDER_TO_NCU.UNIT_01_POWDER_FEEDER_1_STIRRER_SPEED_ACTUAL_LINE_1 := "DB21005_POWDER_FEEDER_PLC_AUX"."INTERLOCKS_PLC_I/O_PF_1_UNIT_01".i_rStirrerActual_Line1;
       "DB7340_NCU_PLC_INTERLOCK".POWDER_TO_NCU.UNIT_01_POWDER_FEEDER_1_HOPPER_TEMPERATURE_ACTUAL_LINE_1 := "DB21005_POWDER_FEEDER_PLC_AUX"."INTERLOCKS_PLC_I/O_PF_1_UNIT_01".i_rHopperTempActual_Line1;
       "DB7340_NCU_PLC_INTERLOCK".POWDER_TO_NCU.UNIT_01_POWDER_FEEDER_1_CARRIER_GAS_ACTUAL_LINE_2 := "DB21005_POWDER_FEEDER_PLC_AUX"."INTERLOCKS_PLC_I/O_PF_1_UNIT_01".i_rCarriergasActual_Line2;
       "DB7340_NCU_PLC_INTERLOCK".POWDER_TO_NCU.UNIT_01_POWDER_FEEDER_1_DISK_SPEED_ACTUAL_LINE_2 := "DB21005_POWDER_FEEDER_PLC_AUX"."INTERLOCKS_PLC_I/O_PF_1_UNIT_01".i_rDiskActual_Line2;
       "DB7340_NCU_PLC_INTERLOCK".POWDER_TO_NCU.UNIT_01_POWDER_FEEDER_1_STIRRER_SPEED_ACTUAL_LINE_2 := "DB21005_POWDER_FEEDER_PLC_AUX"."INTERLOCKS_PLC_I/O_PF_1_UNIT_01".i_rStirrerActual_Line2;
       "DB7340_NCU_PLC_INTERLOCK".POWDER_TO_NCU.UNIT_01_POWDER_FEEDER_1_HOPPER_TEMPERATURE_ACTUAL_LINE_2 := "DB21005_POWDER_FEEDER_PLC_AUX"."INTERLOCKS_PLC_I/O_PF_1_UNIT_01".i_rHopperTempActual_Line2;
   END_IF;
END_REGION

REGION Network 19: UNIT 02 POWDER FEEDER 1 ACTUAL VALUES
   RUNG wire#powerrail
      Contact( "M_ONE" )
      wire#w1
      Move(in := "DB21005_POWDER_FEEDER_PLC_AUX"."INTERLOCKS_PLC_I/O_PF_1_UNIT_02".i_rCarriergasActual_Line1, out1 => "DB7340_NCU_PLC_INTERLOCK".POWDER_TO_NCU.UNIT_02_POWDER_FEEDER_1_CARRIER_GAS_ACTUAL_LINE_1)
      Move(in := "DB21005_POWDER_FEEDER_PLC_AUX"."INTERLOCKS_PLC_I/O_PF_1_UNIT_02".i_rDiskActual_Line1, out1 => "DB7340_NCU_PLC_INTERLOCK".POWDER_TO_NCU.UNIT_02_POWDER_FEEDER_1_DISK_SPEED_ACTUAL_LINE_1)
      Move(in := "DB21005_POWDER_FEEDER_PLC_AUX"."INTERLOCKS_PLC_I/O_PF_1_UNIT_02".i_rStirrerActual_Line1, out1 => "DB7340_NCU_PLC_INTERLOCK".POWDER_TO_NCU.UNIT_02_POWDER_FEEDER_1_STIRRER_SPEED_ACTUAL_LINE_1)
      Move(in := "DB21005_POWDER_FEEDER_PLC_AUX"."INTERLOCKS_PLC_I/O_PF_1_UNIT_02".i_rHopperTempActual_Line1, out1 => "DB7340_NCU_PLC_INTERLOCK".POWDER_TO_NCU.UNIT_02_POWDER_FEEDER_1_HOPPER_TEMPERATURE_ACTUAL_LINE_1)
   END_RUNG
   RUNG wire#w1
      Move(in := "DB21005_POWDER_FEEDER_PLC_AUX"."INTERLOCKS_PLC_I/O_PF_1_UNIT_02".i_rCarriergasActual_Line2, out1 => "DB7340_NCU_PLC_INTERLOCK".POWDER_TO_NCU.UNIT_02_POWDER_FEEDER_1_CARRIER_GAS_ACTUAL_LINE_2)
      Move(in := "DB21005_POWDER_FEEDER_PLC_AUX"."INTERLOCKS_PLC_I/O_PF_1_UNIT_02".i_rDiskActual_Line2, out1 => "DB7340_NCU_PLC_INTERLOCK".POWDER_TO_NCU.UNIT_02_POWDER_FEEDER_1_DISK_SPEED_ACTUAL_LINE_2)
      Move(in := "DB21005_POWDER_FEEDER_PLC_AUX"."INTERLOCKS_PLC_I/O_PF_1_UNIT_02".i_rStirrerActual_Line2, out1 => "DB7340_NCU_PLC_INTERLOCK".POWDER_TO_NCU.UNIT_02_POWDER_FEEDER_1_STIRRER_SPEED_ACTUAL_LINE_2)
      Move(in := "DB21005_POWDER_FEEDER_PLC_AUX"."INTERLOCKS_PLC_I/O_PF_1_UNIT_02".i_rHopperTempActual_Line2, out1 => "DB7340_NCU_PLC_INTERLOCK".POWDER_TO_NCU.UNIT_02_POWDER_FEEDER_1_HOPPER_TEMPERATURE_ACTUAL_LINE_2)
   END_RUNG
   // the same network as SCL:
   IF "M_ONE" THEN
       "DB7340_NCU_PLC_INTERLOCK".POWDER_TO_NCU.UNIT_02_POWDER_FEEDER_1_CARRIER_GAS_ACTUAL_LINE_1 := "DB21005_POWDER_FEEDER_PLC_AUX"."INTERLOCKS_PLC_I/O_PF_1_UNIT_02".i_rCarriergasActual_Line1;
       "DB7340_NCU_PLC_INTERLOCK".POWDER_TO_NCU.UNIT_02_POWDER_FEEDER_1_DISK_SPEED_ACTUAL_LINE_1 := "DB21005_POWDER_FEEDER_PLC_AUX"."INTERLOCKS_PLC_I/O_PF_1_UNIT_02".i_rDiskActual_Line1;
       "DB7340_NCU_PLC_INTERLOCK".POWDER_TO_NCU.UNIT_02_POWDER_FEEDER_1_STIRRER_SPEED_ACTUAL_LINE_1 := "DB21005_POWDER_FEEDER_PLC_AUX"."INTERLOCKS_PLC_I/O_PF_1_UNIT_02".i_rStirrerActual_Line1;
       "DB7340_NCU_PLC_INTERLOCK".POWDER_TO_NCU.UNIT_02_POWDER_FEEDER_1_HOPPER_TEMPERATURE_ACTUAL_LINE_1 := "DB21005_POWDER_FEEDER_PLC_AUX"."INTERLOCKS_PLC_I/O_PF_1_UNIT_02".i_rHopperTempActual_Line1;
       "DB7340_NCU_PLC_INTERLOCK".POWDER_TO_NCU.UNIT_02_POWDER_FEEDER_1_CARRIER_GAS_ACTUAL_LINE_2 := "DB21005_POWDER_FEEDER_PLC_AUX"."INTERLOCKS_PLC_I/O_PF_1_UNIT_02".i_rCarriergasActual_Line2;
       "DB7340_NCU_PLC_INTERLOCK".POWDER_TO_NCU.UNIT_02_POWDER_FEEDER_1_DISK_SPEED_ACTUAL_LINE_2 := "DB21005_POWDER_FEEDER_PLC_AUX"."INTERLOCKS_PLC_I/O_PF_1_UNIT_02".i_rDiskActual_Line2;
       "DB7340_NCU_PLC_INTERLOCK".POWDER_TO_NCU.UNIT_02_POWDER_FEEDER_1_STIRRER_SPEED_ACTUAL_LINE_2 := "DB21005_POWDER_FEEDER_PLC_AUX"."INTERLOCKS_PLC_I/O_PF_1_UNIT_02".i_rStirrerActual_Line2;
       "DB7340_NCU_PLC_INTERLOCK".POWDER_TO_NCU.UNIT_02_POWDER_FEEDER_1_HOPPER_TEMPERATURE_ACTUAL_LINE_2 := "DB21005_POWDER_FEEDER_PLC_AUX"."INTERLOCKS_PLC_I/O_PF_1_UNIT_02".i_rHopperTempActual_Line2;
   END_IF;
END_REGION

REGION Network 20: UNIT 02 POWDER FEEDER 2 ACTUAL VALUES
   RUNG wire#powerrail
      Contact( "M_ONE" )
      wire#w1
      Move(in := "DB21005_POWDER_FEEDER_PLC_AUX"."INTERLOCKS_PLC_I/O_PF_2_UNIT_02".i_rCarriergasActual_Line1, out1 => "DB7340_NCU_PLC_INTERLOCK".POWDER_TO_NCU.UNIT_02_POWDER_FEEDER_2_CARRIER_GAS_ACTUAL_LINE_1)
      Move(in := "DB21005_POWDER_FEEDER_PLC_AUX"."INTERLOCKS_PLC_I/O_PF_2_UNIT_02".i_rDiskActual_Line1, out1 => "DB7340_NCU_PLC_INTERLOCK".POWDER_TO_NCU.UNIT_02_POWDER_FEEDER_2_DISK_SPEED_ACTUAL_LINE_1)
      Move(in := "DB21005_POWDER_FEEDER_PLC_AUX"."INTERLOCKS_PLC_I/O_PF_2_UNIT_02".i_rStirrerActual_Line1, out1 => "DB7340_NCU_PLC_INTERLOCK".POWDER_TO_NCU.UNIT_02_POWDER_FEEDER_2_STIRRER_SPEED_ACTUAL_LINE_1)
      Move(in := "DB21005_POWDER_FEEDER_PLC_AUX"."INTERLOCKS_PLC_I/O_PF_2_UNIT_02".i_rHopperTempActual_Line1, out1 => "DB7340_NCU_PLC_INTERLOCK".POWDER_TO_NCU.UNIT_02_POWDER_FEEDER_2_HOPPER_TEMPERATURE_ACTUAL_LINE_1)
   END_RUNG
   RUNG wire#w1
      Move(in := "DB21005_POWDER_FEEDER_PLC_AUX"."INTERLOCKS_PLC_I/O_PF_2_UNIT_02".i_rCarriergasActual_Line2, out1 => "DB7340_NCU_PLC_INTERLOCK".POWDER_TO_NCU.UNIT_02_POWDER_FEEDER_2_CARRIER_GAS_ACTUAL_LINE_2)
      Move(in := "DB21005_POWDER_FEEDER_PLC_AUX"."INTERLOCKS_PLC_I/O_PF_2_UNIT_02".i_rDiskActual_Line2, out1 => "DB7340_NCU_PLC_INTERLOCK".POWDER_TO_NCU.UNIT_02_POWDER_FEEDER_2_DISK_SPEED_ACTUAL_LINE_2)
      Move(in := "DB21005_POWDER_FEEDER_PLC_AUX"."INTERLOCKS_PLC_I/O_PF_2_UNIT_02".i_rStirrerActual_Line2, out1 => "DB7340_NCU_PLC_INTERLOCK".POWDER_TO_NCU.UNIT_02_POWDER_FEEDER_2_STIRRER_SPEED_ACTUAL_LINE_2)
      Move(in := "DB21005_POWDER_FEEDER_PLC_AUX"."INTERLOCKS_PLC_I/O_PF_2_UNIT_02".i_rHopperTempActual_Line2, out1 => "DB7340_NCU_PLC_INTERLOCK".POWDER_TO_NCU.UNIT_02_POWDER_FEEDER_2_HOPPER_TEMPERATURE_ACTUAL_LINE_2)
   END_RUNG
   // the same network as SCL:
   IF "M_ONE" THEN
       "DB7340_NCU_PLC_INTERLOCK".POWDER_TO_NCU.UNIT_02_POWDER_FEEDER_2_CARRIER_GAS_ACTUAL_LINE_1 := "DB21005_POWDER_FEEDER_PLC_AUX"."INTERLOCKS_PLC_I/O_PF_2_UNIT_02".i_rCarriergasActual_Line1;
       "DB7340_NCU_PLC_INTERLOCK".POWDER_TO_NCU.UNIT_02_POWDER_FEEDER_2_DISK_SPEED_ACTUAL_LINE_1 := "DB21005_POWDER_FEEDER_PLC_AUX"."INTERLOCKS_PLC_I/O_PF_2_UNIT_02".i_rDiskActual_Line1;
       "DB7340_NCU_PLC_INTERLOCK".POWDER_TO_NCU.UNIT_02_POWDER_FEEDER_2_STIRRER_SPEED_ACTUAL_LINE_1 := "DB21005_POWDER_FEEDER_PLC_AUX"."INTERLOCKS_PLC_I/O_PF_2_UNIT_02".i_rStirrerActual_Line1;
       "DB7340_NCU_PLC_INTERLOCK".POWDER_TO_NCU.UNIT_02_POWDER_FEEDER_2_HOPPER_TEMPERATURE_ACTUAL_LINE_1 := "DB21005_POWDER_FEEDER_PLC_AUX"."INTERLOCKS_PLC_I/O_PF_2_UNIT_02".i_rHopperTempActual_Line1;
       "DB7340_NCU_PLC_INTERLOCK".POWDER_TO_NCU.UNIT_02_POWDER_FEEDER_2_CARRIER_GAS_ACTUAL_LINE_2 := "DB21005_POWDER_FEEDER_PLC_AUX"."INTERLOCKS_PLC_I/O_PF_2_UNIT_02".i_rCarriergasActual_Line2;
       "DB7340_NCU_PLC_INTERLOCK".POWDER_TO_NCU.UNIT_02_POWDER_FEEDER_2_DISK_SPEED_ACTUAL_LINE_2 := "DB21005_POWDER_FEEDER_PLC_AUX"."INTERLOCKS_PLC_I/O_PF_2_UNIT_02".i_rDiskActual_Line2;
       "DB7340_NCU_PLC_INTERLOCK".POWDER_TO_NCU.UNIT_02_POWDER_FEEDER_2_STIRRER_SPEED_ACTUAL_LINE_2 := "DB21005_POWDER_FEEDER_PLC_AUX"."INTERLOCKS_PLC_I/O_PF_2_UNIT_02".i_rStirrerActual_Line2;
       "DB7340_NCU_PLC_INTERLOCK".POWDER_TO_NCU.UNIT_02_POWDER_FEEDER_2_HOPPER_TEMPERATURE_ACTUAL_LINE_2 := "DB21005_POWDER_FEEDER_PLC_AUX"."INTERLOCKS_PLC_I/O_PF_2_UNIT_02".i_rHopperTempActual_Line2;
   END_IF;
END_REGION
END_FUNCTION
